FUNCTION_BLOCK FB_UpdateDestination
VAR_INPUT
	fbDestination : FB_DestinationDataStore;
END_VAR
VAR_OUTPUT
END_VAR
VAR
END_VAR

END_FUNCTION_BLOCK

(* stored: Version 1.1.0.1, ProductVersion 3.1.4022.18
   POU FB_UpdateDestination: Id {ab7aee06-55bf-4d9b-8969-b8b26775b1ce}, SpecialFunc None *)
